FUNCTION F_SAFETY_StatusFB_TO_CONNECTIONSHUTDOWN : ST_SAFETY_FBCONNECTIONSHUTDOWN
VAR_INPUT
	stFBStatus						: ST_SAFETY_FBStatus; 	(* Struktura ogolna *)
END_VAR

F_SAFETY_StatusFB_TO_CONNECTIONSHUTDOWN.uStatus.stStatusWords	:= stFBStatus;									(* Przepisanie *)
F_SAFETY_StatusFB_TO_CONNECTIONSHUTDOWN.eState 					:= stFBStatus.BState;							(* Ustawienie enum *)
F_SAFETY_StatusFB_TO_CONNECTIONSHUTDOWN.bGeneralError			:= stFBStatus.wDiagnosis <> 0;					(* General Error *)

END_FUNCTION

(* stored: Version 1.1.0.1, ProductVersion 3.1.4022.12
   POU F_SAFETY_StatusFB_TO_CONNECTIONSHUTDOWN: Id {ee0bdf1a-a4f5-43a1-b9a9-7ca9fbf686f2}, SpecialFunc None *)
